(* IEC 61131-3 sources: SmartHomeNew/SmartHomeNew-main/workspace/system_layer_cleanup/split_scaffold/core_kernel/redundancy_slice, 1 file *)

(* ---- FB_Redundancy_Shadow_Slice_DRAFT.st ---- *)
FUNCTION_BLOCK FB_Redundancy_Shadow_Slice_DRAFT
VAR_INPUT
    VI_System_Time_MS : UDINT;
    VI_Enable : BOOL;
END_VAR
VAR_OUTPUT
    VO_Shadow_Ready : BOOL;
END_VAR
VAR
    // Future target:
    // fbRedundancy : FB_Redundancy_Manager;
END_VAR

// Shadow slice placeholder for redundancy call sequence from PRG_System.
VO_Shadow_Ready := VI_Enable;

END_FUNCTION_BLOCK
